Staubli VAL3: Day3.pjx

--- Day3.pjx ---
Parameters version=s8.13.1Cs9_BS2800 stackSize=5000 millimeterUnit=true
Program file=countBits.pgx
Program file=start.pgx
Program file=stop.pgx
Data file=Day3.dtx
Library alias=util path=Disk://helpers/helpers.pjx
Library alias=math path=Disk://math/math.pjx
Library alias=str path=Disk://string/string.pjx
Type name=lists path=Disk://types/lists/lists.pjx
Type name=lists_num path=Disk://types/lists_num/lists_num.pjx

--- Day3.dtx ---
mdesc mNomSpeed
string sInput
num nInput
lists lResult
  [0]
    string sString
string sCommand
num nValue
string sValue
lists_num lLists_num = {}
num nNum
num nSumPerCol
num nBitResult[12]
num nBitGamma[12]
num nBitEpsilon[12]
num nEpsilon
num nGamma
num nResult
num nDeleteIndex
num nBitOxygen[12]
num nBitCO2[12]
num nResult2

--- start.pgx ---
program start()
  local num l_nNum
  local num l_nElement
  local num l_nCounter
  local num l_nRow
  local num l_nSizeList
  local num l_nDeleteIndex
  local num l_nRESULT
begin

  // read file
  call util:readFile("Disk://input_day3.txt", sInput)
  // sInput[0] = "000011010001"
  // sInput[1] = ""

  call str:splitWord(sInput, lResult)
  // lResult[0].sString[0] = "0"
  // lResult[0].sString[1] = "0"
  // lResult[4].sString[1] = "1"

  // PUZZLE 1

  call countBits(lResult, nSumPerCol)

  for l_nElement = 0 to size(nSumPerCol)-1
    nBitGamma[l_nElement] = sel(nSumPerCol[l_nElement] > size(lResult)/2,1,0)
    nBitEpsilon[l_nElement] = sel(nSumPerCol[l_nElement] > size(lResult)/2,0,1)
  endFor

  call util:bin2dec(nBitEpsilon, nEpsilon)
  call util:bin2dec(nBitGamma, nGamma)

  nResult =  nEpsilon*nGamma

  call util:printNum(nResult)
  // 1131506

  // Puzzle 2

  //
  l_nCounter = 0
  l_nSizeList = size(lResult)
  while l_nSizeList > 1

    call countBits(lResult, nSumPerCol)
    if nSumPerCol[l_nCounter] == size(lResult)/2
      l_nNum = 1
    elseIf nSumPerCol[l_nCounter] > size(lResult)/2
      l_nNum = 1
    else
      l_nNum = 0
    endIf

    // find all rows with l_nNum in cols
    l_nDeleteIndex = 0
    l_nSizeList = size(lResult)
    resize(nDeleteIndex,1,1)
    nDeleteIndex = 0
    for l_nRow = 0 to l_nSizeList-1
      if lResult[l_nRow].sString[l_nCounter]  != toString("",l_nNum)
        append(nDeleteIndex)
        l_nDeleteIndex = l_nDeleteIndex + 1
        nDeleteIndex[l_nDeleteIndex] = l_nRow
      endIf
    endFor
    delete(nDeleteIndex[0])

    // delete unvalid rows:
    for l_nElement = (size(nDeleteIndex)-1) to 0 step -1
      delete(lResult[nDeleteIndex[l_nElement]])
    endFor

    l_nSizeList = size(lResult)
    l_nCounter = l_nCounter+1
  endWhile

  for l_nElement = 0 to 11
    nBitOxygen[l_nElement] = sel(lResult.sString[l_nElement] == "1",1,0)
  endFor

  call util:bin2dec(nBitOxygen, nResult)

  call util:printNum(nResult)

  // Now calc CO2
  call str:splitWord(sInput, lResult)
  l_nCounter = 0
  l_nSizeList = size(lResult)
  while l_nSizeList > 1

    call countBits(lResult, nSumPerCol)
    if nSumPerCol[l_nCounter] == size(lResult)/2
      l_nNum = 0
    elseIf nSumPerCol[l_nCounter] > size(lResult)/2
      l_nNum = 0
    else
      l_nNum = 1
    endIf

    // find all rows with l_nNum in cols
    l_nDeleteIndex = 0
    l_nSizeList = size(lResult)
    resize(nDeleteIndex,1,1)
    nDeleteIndex = 0
    for l_nRow = 0 to l_nSizeList-1
      if lResult[l_nRow].sString[l_nCounter]  != toString("",l_nNum)
        append(nDeleteIndex)
        l_nDeleteIndex = l_nDeleteIndex + 1
        nDeleteIndex[l_nDeleteIndex] = l_nRow
      endIf
    endFor
    delete(nDeleteIndex[0])

    // delete unvalid rows:
    for l_nElement = (size(nDeleteIndex)-1) to 0 step -1
      delete(lResult[nDeleteIndex[l_nElement]])
    endFor

    l_nSizeList = size(lResult)
    l_nCounter = l_nCounter+1
  endWhile

  for l_nElement = 0 to 11
    nBitCO2[l_nElement] = sel(lResult.sString[l_nElement] == "1",1,0)
  endFor

  call util:bin2dec(nBitCO2, nResult2)

  call util:printNum(nResult2)

  // FINALLY: calcualte result

  l_nRESULT = nResult * nResult2

  call util:printNum(l_nRESULT)
  // 7863147
end

--- countBits.pgx ---
program countBits(lists& x_lInput[], num& x_nResult[])
  local num l_nElement
  local num l_nBits
begin

  resize(x_nResult,1,1)
  x_nResult[0] = 0
  resize(x_nResult,1,12)

  for l_nBits = 0 to 11
    for l_nElement = 0 to size(x_lInput)-1
      call util:vec2num(x_lInput[l_nElement].sString[l_nBits], nNum)
      x_nResult[l_nBits] = x_nResult[l_nBits] + nNum
    endFor
  endFor


end
